// TIA Portal project "Contadores" (V17)

(* hardware
DEVICE "S7-1500/ET200MP station_1"  S7-1500 station
   slot 0: "Rail_0"  Rack  6ES7 590-1***0-0AA0
   slot 1: "PLC_1"  CPU 1511-1 PN  6ES7 511-1AK00-0AB0  V1.8
      slot 3: "CPU display_1"  6ES7591-1AA00-0AA0
      slot 32768: "PROFINET interface_1"  X1
         slot 32769: "Port_1"  X1 P1
         slot 32770: "Port_2"  X1 P2
*)

// ===== PLC "PLC_1"  CPU 1511-1 PN =====

VAR_GLOBAL   // PLC tag table "Default tag table"
   "Tag_1" AT %I0.2 : Bool;
   "Tag_2" AT %C5 : Counter;
   "Tag_3" AT %I3.0 : Bool;
   "Tag_4" AT %E0.0 : Bool;
   "Tag_5" AT %M0.0 : Bool;
   "Tag_6" AT %Z1 : Counter;
   "Tag_7" AT %E0.1 : Bool;
   "Tag_8" AT %E0.3 : Bool;
   "Tag_9" AT %A0.0 : Bool;
   "Tag_10" AT %A0.1 : Bool;
   "Tag_11" AT %E0.4 : Bool;
   "Tag_12" AT %Z2 : Counter;
   "Tag_13" AT %E1.0 : Bool;
   "Tag_14" AT %M1.0 : Bool;
   "Tag_15" AT %E1.1 : Bool;
   "Tag_16" AT %A1.0 : Bool;
   "Tag_17" AT %A1.1 : Bool;
   "Tag_18" AT %E1.2 : Bool;
   "Tag_19" AT %E2.0 : Bool;
   "Tag_20" AT %Z3 : Counter;
   "Tag_21" AT %M2.0 : Bool;
   "Tag_22" AT %A2.1 : Bool;
   "Tag_23" AT %A2.0 : Bool;
   "Tag_24" AT %A2.2 : Bool;
   "Tag_25" AT %A2.3 : Bool;
   "Tag_26" AT %A0.4 : Bool;
   "Tag_27" AT %E2.1 : Bool;
   "Tag_28" AT %E2.2 : Bool;
   "Clock_Byte" AT %MB5 : Byte;
   "Clock_10Hz" AT %M5.0 : Bool;
   "Clock_5Hz" AT %M5.1 : Bool;
   "Clock_2.5Hz" AT %M5.2 : Bool;
   "Clock_2Hz" AT %M5.3 : Bool;
   "Clock_1.25Hz" AT %M5.4 : Bool;
   "Clock_1Hz" AT %M5.5 : Bool;
   "Clock_0.625Hz" AT %M5.6 : Bool;
   "Clock_0.5Hz" AT %M5.7 : Bool;
   "Tag_29" AT %Z4 : Counter;
   "Tag_30" AT %A3.0 : Bool;
END_VAR

ORGANIZATION_BLOCK "Main"   // OB1, LAD, ProgramCycle
TITLE = "Main Program Sweep (Cycle)"
{ S7_Optimized_Access := 'TRUE' }
VERSION : 0.1
   VAR_INPUT
      Initial_Call : Bool;   // Initial call of this OB
      Remanence : Bool;   // =True, if remanent data are available
   END_VAR
BEGIN

REGION Network 2 (STL)
         A     "Tag_4";
         AN    "Tag_5";
         L     C#10;
         S     "Tag_6";
         S     "Tag_5";

         A     "Tag_7";
         AN    "Tag_5";
         L     C#20;
         S     "Tag_6";
         S     "Tag_5";

         A     "Tag_1";
         AN    "Tag_5";
         L     c#20;
         S     "Tag_6";
         S     "Tag_5";


         A     "Tag_5";  // INDICA CONTADOR CARGADO
         A     "Tag_8";  // ENTRADA DIGITAL PARA RESTAR AL CONTADOR
         CD    "Tag_6";

         AN    "Tag_6";  // CONSULTA CONTADOR
         =     "Tag_9";  // INDICA CONTADOR A CERO

         L     "Tag_6";
         L     9;
         >I;
         =     "Tag_10";  // INDICA QUE EL CONTADOR ES MAYOR A 9

         A     "Tag_11";  // REINICIAR CONTADOR Y MARCA
         R     "Tag_6";
         R     "Tag_5";
END_REGION

REGION Network 3 (STL)
         A     "Tag_13";
         L     C#10;
         S     "Tag_12";  // CONTADOR Z2
         S     "Tag_14";  // MARCA DE ESTADO

         A     "Tag_15";  //ENTRADA DE COCHE
         A     "Tag_14";  //CONTADOR CARGADO
         A     "Tag_12";
         =     "Tag_16";  //LEVANTAR PLUMA
         CD    "Tag_12";  //RESTAR UNO CUANDO ENTRA COCHE


         A     "Tag_12";
         =     "Tag_17";  //ENCENDER PLAZA LIBRE

         A     "Tag_18";  //CELULA DE SALIDA
         CU    "Tag_12";  //SUMAR UNO CUANDO SALE COCHE
END_REGION

REGION Network 4 (STL)
   //ALMACEN DE 10
         A     "Tag_19";  // CARGA DE ALMACEN
         L     C#10;
         S     "Tag_20";  // SETEAMOS CONTADOR


         AN    "Tag_20";  // vacio
         =     "Tag_23";  // ENCENDIDO DE LINEA

         A     "Tag_20";  //NO VACIO
         AN(;
         L     "Tag_20";  // Y NO LLENO
         L     10;
         >=I;
         );
         =     "Tag_22";  //ENDENDIDO DE LINEA

         L     "Tag_20";
         L     5;
         >=I;
         =     "Tag_24";  // AL 50%

         L     "Tag_20";
         L     9;
         >=I;
         =     "Tag_25";  //MAS DEL 90%

         L     "Tag_20";
         L     10;
         >=I;
         =     "Tag_26";  // LLENO


         A     "Tag_27";
         CD    "Tag_20";

         A     "Tag_28";
         CU    "Tag_20";
END_REGION

REGION Network 5 (STL)
   // CONTADOR CON MARCAS
         A     "Tag_3";
         L     C#50;
         S     "Tag_29";

         A     "Clock_1Hz";
         CD    "Tag_29";

         AN    "Tag_29";
         =     "Tag_30";
END_REGION
END_ORGANIZATION_BLOCK